PROGRAM Manual_POU
VAR
	fbGeneralAxis:ARRAY [1..6]OF FB_AxisGeneral;
	Clear							:ST_HMIAxieControl;
	HMIAxis_Box,HMIAxis_Dual1,HMIAxis_Dual2,HMIAxis_flyin,HMIAxis_load1,HMIAxis_load2				:ST_HMIAxieControl;
	wAxisNumb,wControlNumb,nChangeStep	:INT;
	tmrChangeMode			:TON;
	wTemp,i		:INT;
	bHMI_VerticalRoller , bHMI_VerticalBelt	:BOOL;
	bHMI_UnboxingInitial	,bHMI_UnboxingInitialDone,bHMI_UnboxingStart,bHMI_UnboxingDone:BOOL;
	bDualGearIn,bDualGearOut	:BOOL;
	MC_GearIn,MC_GearInload:MC_GearIn;
	MC_GearOut,MC_GearOutload:MC_GearOut;
	A1TouchPos,A2TouchPos					:ARRAY [1..5] OF LREAL;
	tempA1,tempA2	:LREAL;
	fbMC_UngroupAllAxes	: MC_UngroupAllAxes;
	fbMC_GroupDisable	: MC_GroupDisable;
	
END_VAR

Roller();
Axis();

ACTION Axis:
fbGeneralAxis[1](Axis:= Axis_FlyIn,HmiPanel:= HMIAxis_flyin);
fbGeneralAxis[2](Axis:= Axis_DualServo1,HmiPanel:= HMIAxis_Dual1);
fbGeneralAxis[3](Axis:= Axis_DualServo2,HmiPanel:= HMIAxis_Dual2);
fbGeneralAxis[4](Axis:= Axis_BoxPullOut,HmiPanel:= HMIAxis_Box,i_homecam:= NOT Sen_AxisBoxORG);	
fbGeneralAxis[5](Axis:= Axis_load1,HmiPanel:= HMIAxis_load1);
fbGeneralAxis[6](Axis:= Axis_load2,HmiPanel:= HMIAxis_load2);

MC_GearIn(
	Master:= Axis_DualServo1, 
	Slave:= Axis_DualServo2, 
	Execute:= bDualGearIn, 
	RatioNumerator:= , 
	RatioDenominator:= , 
	Acceleration:= , 
	Deceleration:= , 
	Jerk:= , 
	BufferMode:= , 
	Options:= , 
	InGear=> , 
	Busy=> , 
	Active=> , 
	CommandAborted=> , 
	Error=> , 
	ErrorID=> );

MC_GearOut(
	Slave:= Axis_DualServo2, 
	Execute:= bDualGearOut, 
);		

MC_GearInload(
	Master:= Axis_load1, 
	Slave:= Axis_load2, 
	Execute:= , 
	RatioNumerator:= , 
	RatioDenominator:= , 
	Acceleration:= , 
	Deceleration:= , 
	Jerk:= , 
	BufferMode:= , 
	Options:= , 
	InGear=> , 
	Busy=> , 
	Active=> , 
	CommandAborted=> , 
	Error=> , 
	ErrorID=> );

MC_GearOutload(
	Slave:= Axis_load2, 
	Execute:= , 
);		
UngroupAllAxes();
END_ACTION

ACTION Roller:
IF bHMI_VerticalRoller THEN
	AssRoller.Roller();	
END_IF

IF bHMI_VerticalBelt THEN
	AssRoller.Belt();	
END_IF
END_ACTION

ACTION Seizure:
(*
tmrChangeMode(PT:=T#1S);



CASE wControlNumb OF
	0:
		fbGeneralAxis[1](Axis:= Axis_FlyIn,HmiPanel:= HMIControlAxis);
	1:
		fbGeneralAxis[2](Axis:= Axis_Conv1,HmiPanel:= HMIControlAxis);
	2:
		fbGeneralAxis[3](Axis:= Axis_Conv2,HmiPanel:= HMIControlAxis);
	3:
		fbGeneralAxis[4](Axis:= Axis_BoxPullOut,HmiPanel:= HMIControlAxis);	
	4:
		fbGeneralAxis[5](Axis:= Axis_Unload1,HmiPanel:= HMIControlAxis);
	5:
		fbGeneralAxis[6](Axis:= Axis_Unload2,HmiPanel:= HMIControlAxis);
END_CASE
CASE nChangeStep OF
	0:
		IF wTemp<> wAxisNumb THEN
			nChangeStep	 := 5 ;
		END_IF; 

	5:
		HMIControlAxis:= Clear;
		tmrChangeMode(IN:= TRUE,PT:=T#1S);
		IF tmrChangeMode.Q THEN
			tmrChangeMode(IN:= FALSE);
			wControlNumb	:= wAxisNumb;
			nChangeStep	 	:= 0 ;
		END_IF


END_CASE


wTemp	:= wAxisNumb ;
*)
END_ACTION

METHOD UngroupAllAxes : BOOL
fbMC_GroupDisable(
	AxesGroup:= DualGroupRef, 
	Execute:= , 
	Done=> , 
	Busy=> , 
	Error=> , 
	ErrorId=> );	

fbMC_UngroupAllAxes(
	AxesGroup:= DualGroupRef, 
	Execute:= fbMC_GroupDisable.Done, 
	Done=> , 
	Busy=> , 
	Error=> , 
	ErrorId=> );	
	
UngroupAllAxes :=fbMC_UngroupAllAxes.Done AND fbMC_GroupDisable.Done;
END_METHOD

END_PROGRAM

(* stored: Version 1.1.0.1, ProductVersion 3.1.4024.16
   POU Manual_POU: Id {48250a18-44d0-49bc-8f62-7b4b94f75257}, SpecialFunc None
   Action Axis: Id {a8c6ee8a-1977-47ca-9ffa-1eff20488e7a}
   Action Roller: Id {83b3b19c-1248-4507-9ca7-e03f600c5e09}
   Action Seizure: Id {dfe7ba06-b60b-4710-88d0-89aa4fe757ba}
   Method UngroupAllAxes: Id {46f9945f-0b23-4d86-9aa0-67027dd84466} *)
